// SIMATIC S7-200 SMART project (STEP 7-Micro/WIN SMART), CPU SR40

ORGANIZATION_BLOCK MAIN:OB1
TITLE=程序注释
BEGIN
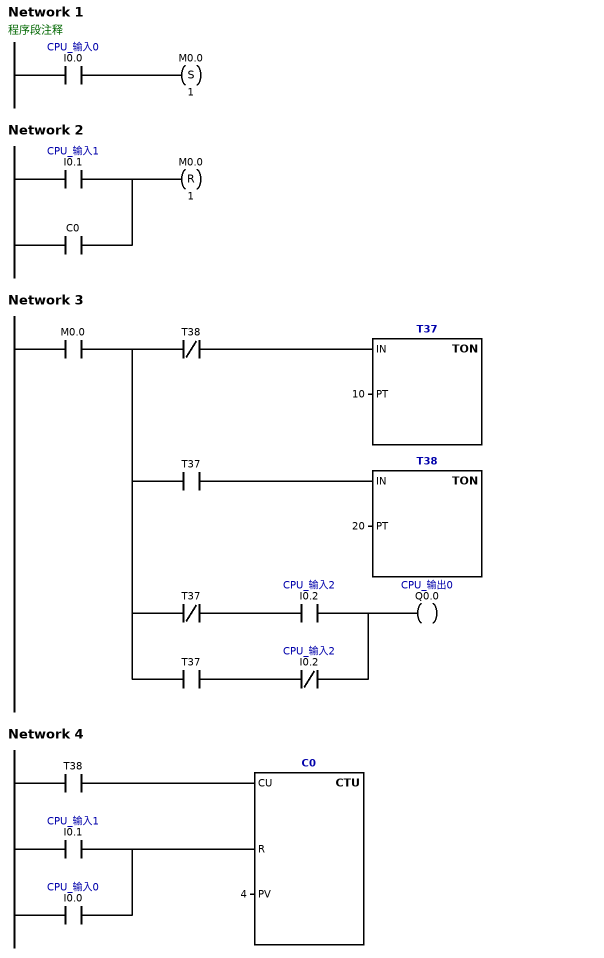
Network 1
// 程序段注释
LD     CPU_输入0:I0.0
S      M0.0, 1
Network 2
LD     CPU_输入1:I0.1
O      C0
R      M0.0, 1
Network 3
LD     M0.0
LPS
AN     T38
TON    T37, 10
LRD
A      T37
TON    T38, 20
LPP
LDN    T37
A      CPU_输入2:I0.2
LD     T37
AN     CPU_输入2:I0.2
OLD
ALD
=      CPU_输出0:Q0.0
Network 4
// (network saved uncompiled; LAD cells follow)
// row 0: c0 -| |- T38  c1 --  c2 [CTU C0 CU:=power@row0, R:=power@row1, PV:=4]
// row 1: c0 -| |- CPU_输入1:I0.1 v  c1 --  c2 [box]
// row 2: c0 -| |- CPU_输入0:I0.0 ^  c2 [box]
END_ORGANIZATION_BLOCK
